// TIA Portal V19 export
DATA_BLOCK "DB_PNOZ_Comm"   // DB360
{ S7_Optimized_Access := 'FALSE' }
// stored: AutoNumber false
   VAR
      Global_Status : Int;   // 0: OFF; 1: CONNECT; 2: WRITE; 3: READ; 4: DISCONNECT; 5: ERROR
      connection : Struct
         activate : Bool := TRUE;
         established : Bool;   // E
      END_STRUCT;
      CONNECT : Struct
         Request : Bool := TRUE;
         Done : Bool;
         Busy : Bool;
         Error : Bool;
         ID : Word := WORD#16#0002;
         Status : Word;
      END_STRUCT;
      SEND : Struct
         Request : Bool;
         Done : Bool;
         Busy : Bool;
         Error : Bool;
         ID : Word := WORD#16#0002;
         Status : Word;
         Length : UDInt := 43;
      END_STRUCT;
      RECEIVE : Struct
         EN_R : Bool := TRUE;
         ADHOC : Bool := FALSE;
         NDR : Bool := TRUE;
         Busy : Bool;
         Error : Bool;
         ID : Word := WORD#16#0002;
         Status : Word;
         Length : UDInt := 43;
         Receive_Length : UDInt := 43;
      END_STRUCT;
      DISCONNECT : Struct
         Request : Bool;
         Done : Bool;
         Busy : Bool;
         Error : Bool;
         ID : Word;
         Status : Word;
      END_STRUCT;
      Connection_Param { S7_SetPoint := 'True'} : "PNOZ Comm";
   END_VAR
BEGIN
   Connection_Param.local_device_id := BYTE#16#02;
   Connection_Param.rem_staddr[1] := BYTE#16#0A;
   Connection_Param.rem_staddr[2] := BYTE#16#94;
   Connection_Param.rem_staddr[3] := B#16#22;
   Connection_Param.rem_staddr[4] := BYTE#16#46;
END_DATA_BLOCK
